(* IEC 61131-3 sources: plc_generation_empirical_study/datasets/packages/internal_v0_1_precalibration_20260810/qualification_only/C04_M01_falling_edge_pulse/negative_control, 1 file *)

(* ---- NC1.st ---- *)
FUNCTION_BLOCK C04_M01_falling_edge_pulse
VAR_INPUT
    Signal : BOOL;
    Arm : BOOL;
END_VAR
VAR_OUTPUT
    Pulse : BOOL;
    Armed : BOOL;
END_VAR
VAR
    PrevSignal : BOOL := TRUE;
END_VAR

Pulse := Arm AND (NOT Signal) AND PrevSignal;
Armed := Arm;
PrevSignal := Signal;

END_FUNCTION_BLOCK
